TYPE (* A Structure with 2 Bits *)
  (* Version 1.0, 2024-02-21, franz *)
  st2bits : STRUCT
    b0 : BOOL; (* BIT 00 *)
    b1 : BOOL; (* BIT 01 *)
  END_STRUCT;
END_TYPE
